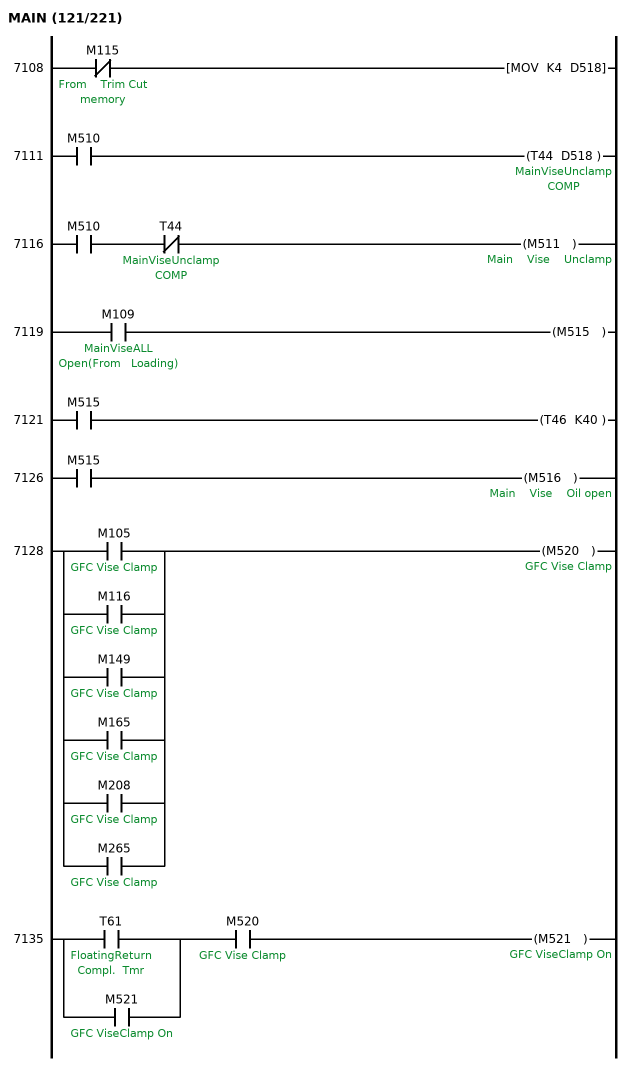
[picture p120: ladder of MAIN, rungs at steps 7108 to 7135]
7108  LDI     M115  ; From    Trim Cut memory
      MOV     K4 D518
7111  LD      M510
      OUT     T44 D518  ; MainViseUnclamp COMP
7116  LD      M510
      ANI     T44  ; MainViseUnclamp COMP
      OUT     M511  ; Main    Vise    Unclamp
7119  LD      M109  ; MainViseALL Open(From   Loading)
      OUT     M515
7121  LD      M515
      OUT     T46 K40
7126  LD      M515
      OUT     M516  ; Main    Vise    Oil open
7128  LD      M105  ; GFC Vise Clamp
      OR      M116  ; GFC Vise Clamp
      OR      M149  ; GFC Vise Clamp
      OR      M165  ; GFC Vise Clamp
      OR      M208  ; GFC Vise Clamp
      OR      M265  ; GFC Vise Clamp
      OUT     M520  ; GFC Vise Clamp
7135  LD      T61  ; FloatingReturn  Compl.  Tmr
      OR      M521  ; GFC ViseClamp On
      AND     M520  ; GFC Vise Clamp
      OUT     M521  ; GFC ViseClamp On
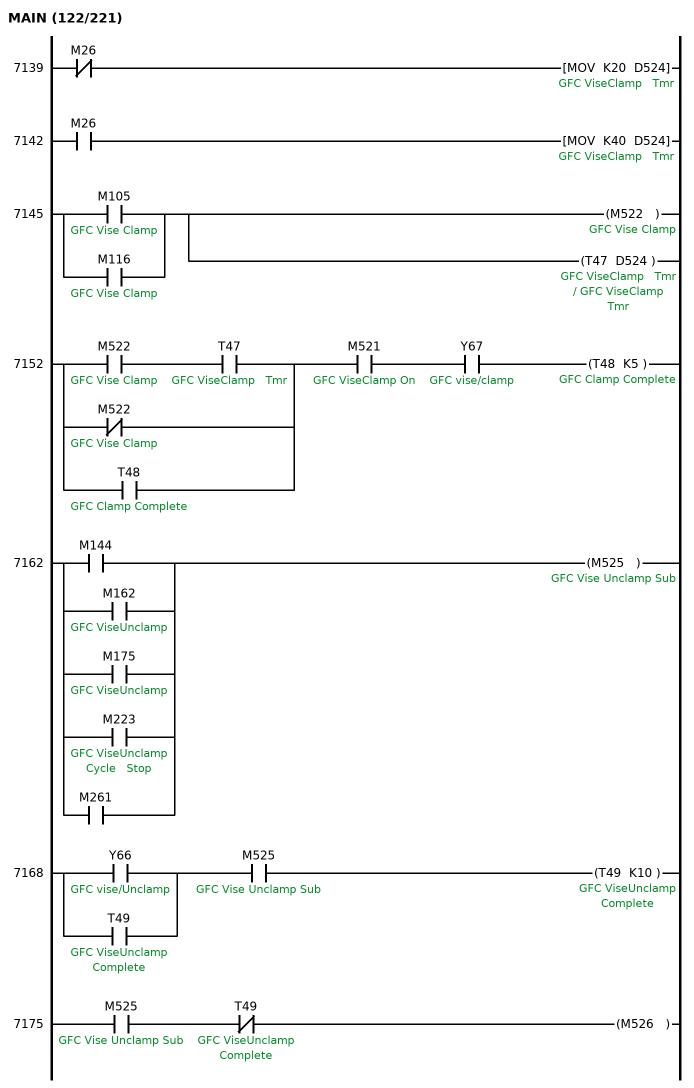
7139  LDI     M26
      MOV     K20 D524  ; GFC ViseClamp   Tmr
7142  LD      M26
      MOV     K40 D524
7145  LD      M105  ; GFC Vise Clamp
      OR      M116  ; GFC Vise Clamp
      OUT     M522  ; GFC Vise Clamp
      OUT     T47 D524  ; GFC ViseClamp   Tmr / GFC ViseClamp   Tmr
7152  LD      M522  ; GFC Vise Clamp
      AND     T47  ; GFC ViseClamp   Tmr
      ORI     M522  ; GFC Vise Clamp
      OR      T48  ; GFC Clamp Complete
      AND     M521  ; GFC ViseClamp On
      AND     Y67  ; GFC vise/clamp
      OUT     T48 K5  ; GFC Clamp Complete
7162  LD      M144
      OR      M162  ; GFC ViseUnclamp
      OR      M175  ; GFC ViseUnclamp
      OR      M223  ; GFC ViseUnclamp Cycle   Stop
      OR      M261
      OUT     M525  ; GFC Vise Unclamp Sub
7168  LD      Y66  ; GFC vise/Unclamp
      OR      T49  ; GFC ViseUnclamp Complete
      AND     M525  ; GFC Vise Unclamp Sub
      OUT     T49 K10  ; GFC ViseUnclamp Complete
7175  LD      M525  ; GFC Vise Unclamp Sub
      ANI     T49  ; GFC ViseUnclamp Complete
      OUT     M526
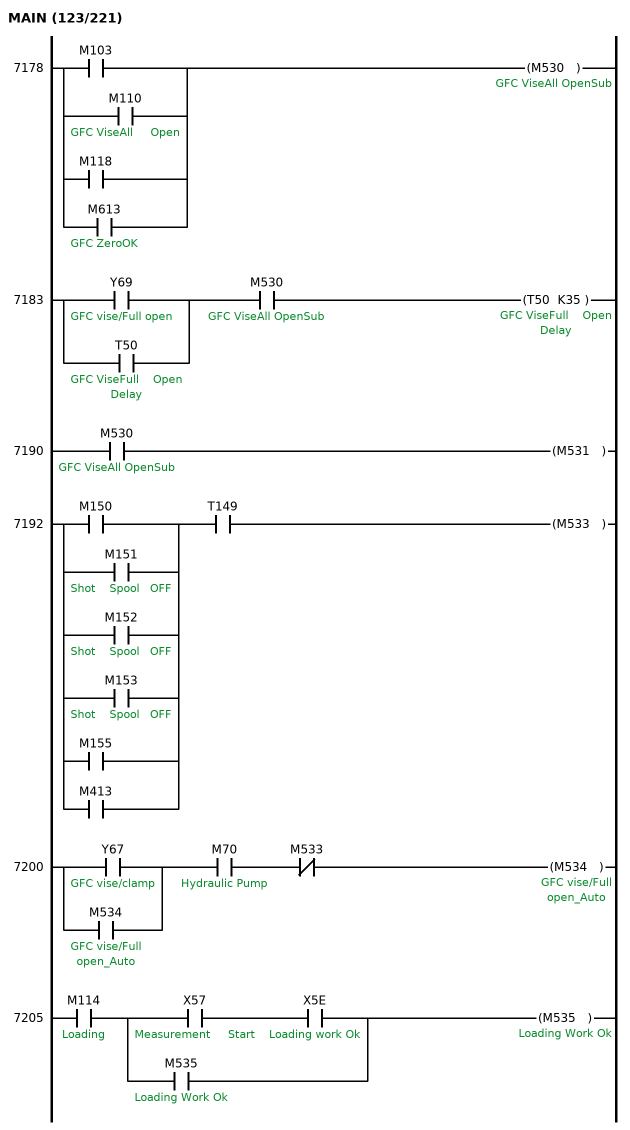
7178  LD      M103
      OR      M110  ; GFC ViseAll     Open
      OR      M118
      OR      M613  ; GFC ZeroOK
      OUT     M530  ; GFC ViseAll OpenSub
7183  LD      Y69  ; GFC vise/Full open
      OR      T50  ; GFC ViseFull    Open    Delay
      AND     M530  ; GFC ViseAll OpenSub
      OUT     T50 K35  ; GFC ViseFull    Open    Delay
7190  LD      M530  ; GFC ViseAll OpenSub
      OUT     M531
7192  LD      M150
      OR      M151  ; Shot    Spool   OFF
      OR      M152  ; Shot    Spool   OFF
      OR      M153  ; Shot    Spool   OFF
      OR      M155
      OR      M413
      AND     T149
      OUT     M533
7200  LD      Y67  ; GFC vise/clamp
      OR      M534  ; GFC vise/Full open_Auto
      AND     M70  ; Hydraulic Pump
      ANI     M533
      OUT     M534  ; GFC vise/Full open_Auto
7205  LD      M114  ; Loading
      LD      X57  ; Measurement     Start
      AND     X5E  ; Loading work Ok
      OR      M535  ; Loading Work Ok
      ANB
      OUT     M535  ; Loading Work Ok
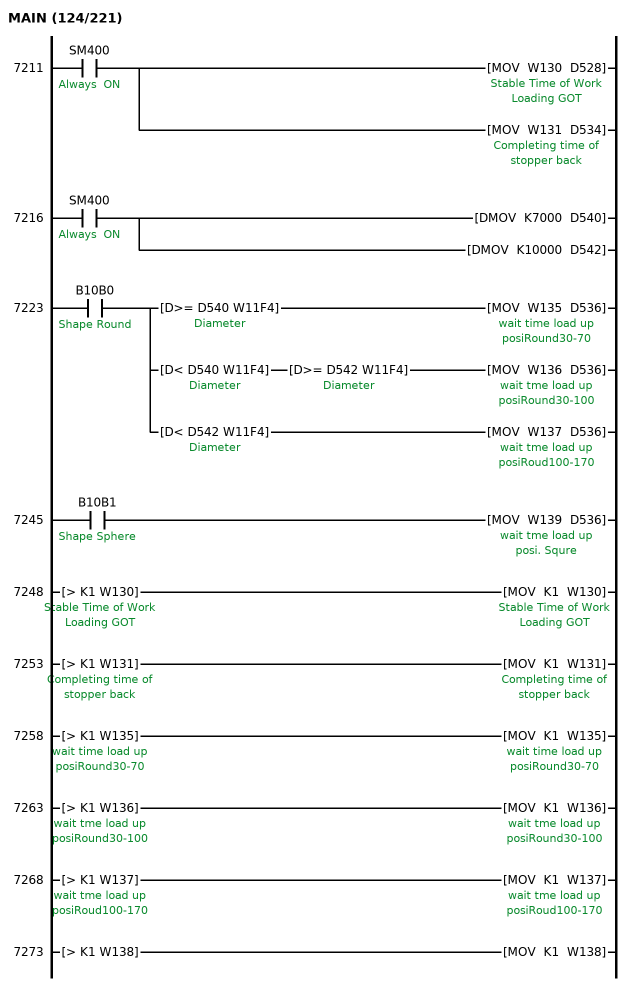
7211  LD      SM400  ; Always  ON
      MOV     W130 D528
      MOV     W131 D534  ; Completing time of stopper back
7216  LD      SM400  ; Always  ON
      DMOV    K7000 D540
      DMOV    K10000 D542
7223  LD      B10B0  ; Shape Round
      MPS
      ANDD>=  D540 W11F4  ; Diameter
      MOV     W135 D536  ; wait time load up posiRound30-70
      MRD
      ANDD<   D540 W11F4  ; Diameter
      ANDD>=  D542 W11F4  ; Diameter
      MOV     W136 D536  ; wait tme load up posiRound30-100
      MPP
      ANDD<   D542 W11F4  ; Diameter
      MOV     W137 D536  ; wait tme load up posiRoud100-170
7245  LD      B10B1  ; Shape Sphere
      MOV     W139 D536  ; wait tme load up posi. Squre
7248  LD>     K1 W130  ; Stable Time of Work Loading GOT
      MOV     K1 W130
7253  LD>     K1 W131  ; Completing time of stopper back
      MOV     K1 W131
7258  LD>     K1 W135  ; wait time load up posiRound30-70
      MOV     K1 W135
7263  LD>     K1 W136  ; wait tme load up posiRound30-100
      MOV     K1 W136
7268  LD>     K1 W137  ; wait tme load up posiRoud100-170
      MOV     K1 W137
7273  LD>     K1 W138
      MOV     K1 W138
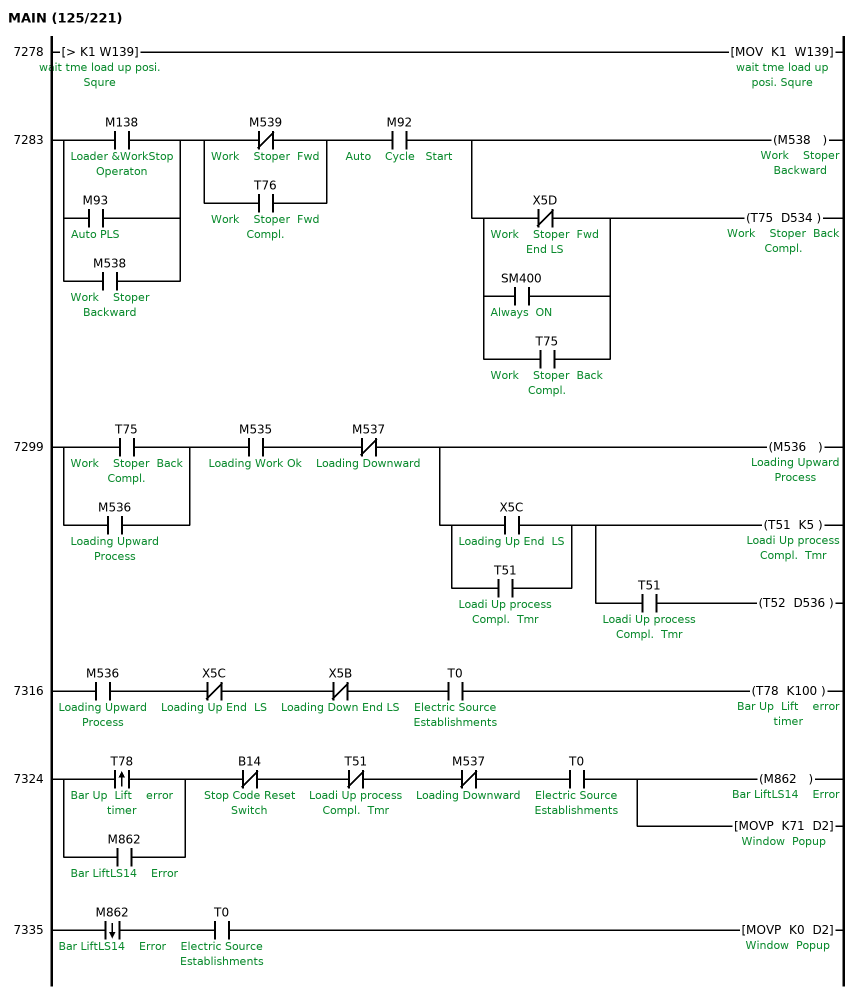
7278  LD>     K1 W139  ; wait tme load up posi. Squre
      MOV     K1 W139
7283  LD      M138  ; Loader &WorkStopOperaton
      OR      M93  ; Auto PLS
      OR      M538  ; Work    Stoper  Backward
      LDI     M539  ; Work    Stoper  Fwd
      OR      T76  ; Work    Stoper  Fwd     Compl.
      ANB
      AND     M92  ; Auto    Cycle   Start
      OUT     M538  ; Work    Stoper  Backward
      LDI     X5D  ; Work    Stoper  Fwd End LS
      OR      SM400  ; Always  ON
      OR      T75  ; Work    Stoper  Back    Compl.
      ANB
      OUT     T75 D534  ; Work    Stoper  Back    Compl.
7299  LD      T75  ; Work    Stoper  Back    Compl.
      OR      M536  ; Loading Upward  Process
      AND     M535  ; Loading Work Ok
      ANI     M537  ; Loading Downward
      OUT     M536  ; Loading Upward  Process
      LD      X5C  ; Loading Up End  LS
      OR      T51  ; Loadi Up process Compl.  Tmr
      ANB
      OUT     T51 K5  ; Loadi Up process Compl.  Tmr
      AND     T51  ; Loadi Up process Compl.  Tmr
      OUT     T52 D536
7316  LD      M536  ; Loading Upward  Process
      ANI     X5C  ; Loading Up End  LS
      ANI     X5B  ; Loading Down End LS
      AND     T0  ; Electric Source Establishments
      OUT     T78 K100  ; Bar Up  Lift    error   timer
7324  LDP     T78  ; Bar Up  Lift    error   timer
      OR      M862  ; Bar LiftLS14    Error
      ANI     B14  ; Stop Code Reset Switch
      ANI     T51  ; Loadi Up process Compl.  Tmr
      ANI     M537  ; Loading Downward
      AND     T0  ; Electric Source Establishments
      OUT     M862  ; Bar LiftLS14    Error
      MOVP    K71 D2  ; Window  Popup
7335  LDF     M862  ; Bar LiftLS14    Error
      AND     T0  ; Electric Source Establishments
      MOVP    K0 D2
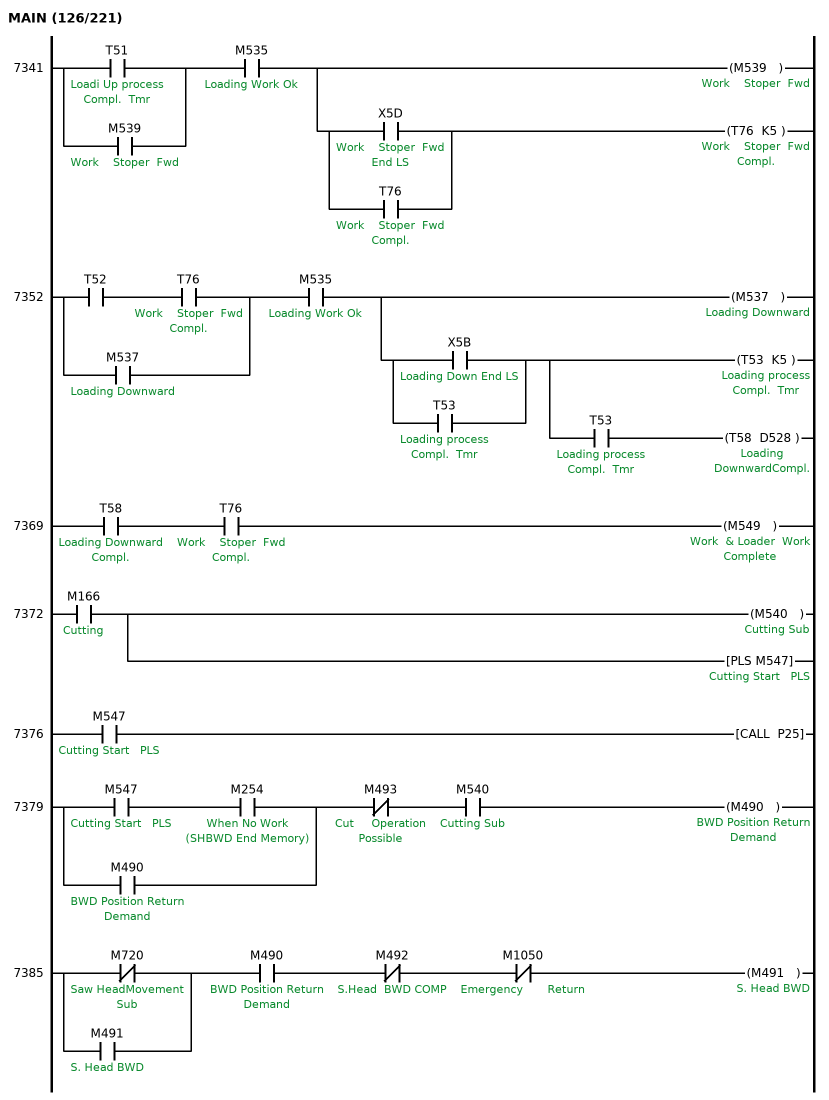
7341  LD      T51  ; Loadi Up process Compl.  Tmr
      OR      M539  ; Work    Stoper  Fwd
      AND     M535  ; Loading Work Ok
      OUT     M539  ; Work    Stoper  Fwd
      LD      X5D  ; Work    Stoper  Fwd End LS
      OR      T76  ; Work    Stoper  Fwd     Compl.
      ANB
      OUT     T76 K5  ; Work    Stoper  Fwd     Compl.
7352  LD      T52
      AND     T76  ; Work    Stoper  Fwd     Compl.
      OR      M537  ; Loading Downward
      AND     M535  ; Loading Work Ok
      OUT     M537  ; Loading Downward
      LD      X5B  ; Loading Down End LS
      OR      T53  ; Loading process Compl.  Tmr
      ANB
      OUT     T53 K5  ; Loading process Compl.  Tmr
      AND     T53  ; Loading process Compl.  Tmr
      OUT     T58 D528  ; Loading DownwardCompl.
7369  LD      T58  ; Loading DownwardCompl.
      AND     T76  ; Work    Stoper  Fwd     Compl.
      OUT     M549  ; Work  & Loader  Work Complete
7372  LD      M166  ; Cutting
      OUT     M540  ; Cutting Sub
      PLS     M547  ; Cutting Start   PLS
7376  LD      M547  ; Cutting Start   PLS
      CALL    P25
7379  LD      M547  ; Cutting Start   PLS
      AND     M254  ; When No Work (SHBWD End Memory)
      OR      M490  ; BWD Position Return Demand
      ANI     M493  ; Cut     Operation       Possible
      AND     M540  ; Cutting Sub
      OUT     M490  ; BWD Position Return Demand
7385  LDI     M720  ; Saw HeadMovementSub
      OR      M491  ; S. Head BWD
      AND     M490  ; BWD Position Return Demand
      ANI     M492  ; S.Head  BWD COMP
      ANI     M1050  ; Emergency       Return
      OUT     M491  ; S. Head BWD
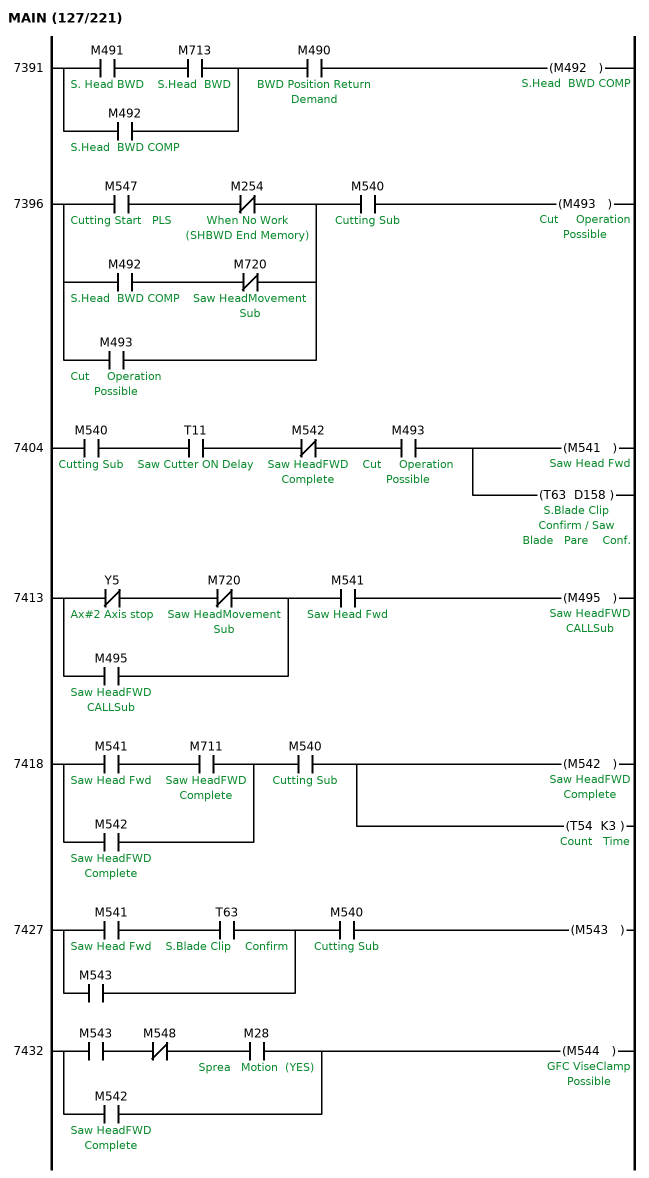
7391  LD      M491  ; S. Head BWD
      AND     M713  ; S.Head  BWD
      OR      M492  ; S.Head  BWD COMP
      AND     M490  ; BWD Position Return Demand
      OUT     M492  ; S.Head  BWD COMP
7396  LD      M547  ; Cutting Start   PLS
      ANI     M254  ; When No Work (SHBWD End Memory)
      LD      M492  ; S.Head  BWD COMP
      ANI     M720  ; Saw HeadMovementSub
      ORB
      OR      M493  ; Cut     Operation       Possible
      AND     M540  ; Cutting Sub
      OUT     M493  ; Cut     Operation       Possible
7404  LD      M540  ; Cutting Sub
      AND     T11  ; Saw Cutter ON Delay
      ANI     M542  ; Saw HeadFWD     Complete
      AND     M493  ; Cut     Operation       Possible
      OUT     M541  ; Saw Head Fwd
      OUT     T63 D158  ; S.Blade Clip    Confirm / Saw     Blade   Pare    Conf.
7413  LDI     Y5  ; Ax#2 Axis stop
      ANI     M720  ; Saw HeadMovementSub
      OR      M495  ; Saw HeadFWD CALLSub
      AND     M541  ; Saw Head Fwd
      OUT     M495  ; Saw HeadFWD CALLSub
7418  LD      M541  ; Saw Head Fwd
      AND     M711  ; Saw HeadFWD     Complete
      OR      M542  ; Saw HeadFWD     Complete
      AND     M540  ; Cutting Sub
      OUT     M542  ; Saw HeadFWD     Complete
      OUT     T54 K3  ; Count   Time
7427  LD      M541  ; Saw Head Fwd
      AND     T63  ; S.Blade Clip    Confirm
      OR      M543
      AND     M540  ; Cutting Sub
      OUT     M543
7432  LD      M543
      ANI     M548
      AND     M28  ; Sprea   Motion  (YES)
      OR      M542  ; Saw HeadFWD     Complete
      OUT     M544  ; GFC ViseClamp   Possible
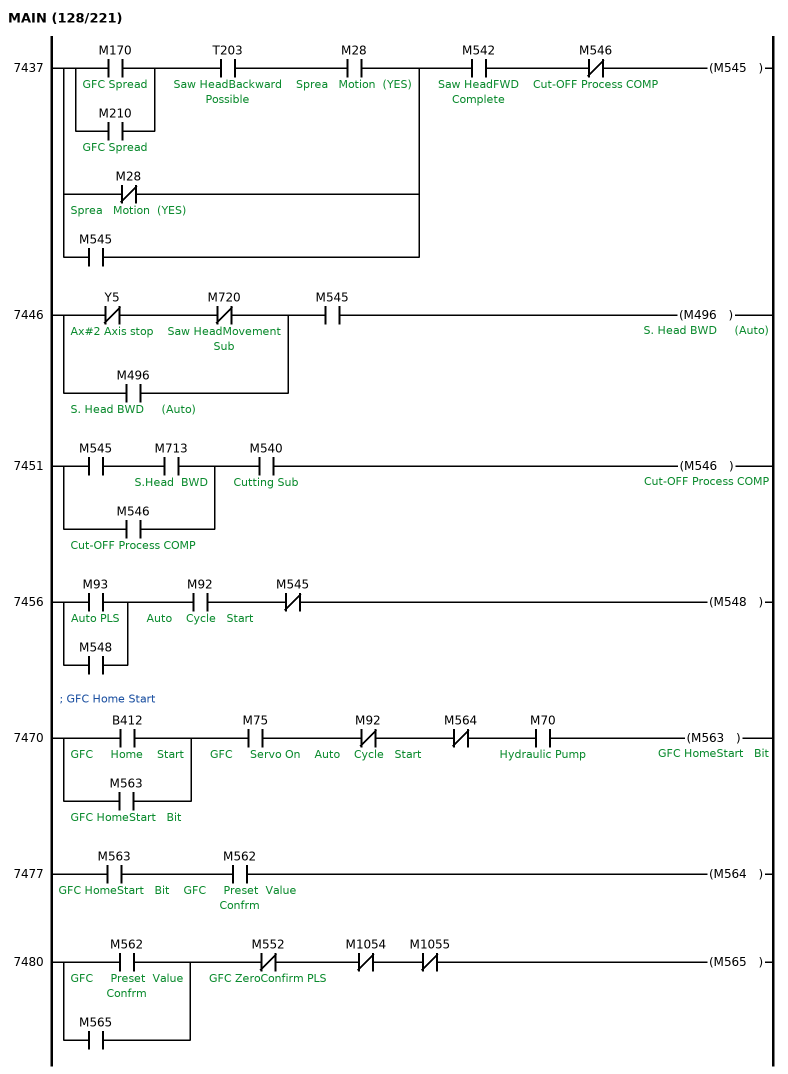
7437  LD      M170  ; GFC Spread
      OR      M210  ; GFC Spread
      AND     T203  ; Saw HeadBackwardPossible
      AND     M28  ; Sprea   Motion  (YES)
      ORI     M28  ; Sprea   Motion  (YES)
      OR      M545
      AND     M542  ; Saw HeadFWD     Complete
      ANI     M546  ; Cut-OFF Process COMP
      OUT     M545
7446  LDI     Y5  ; Ax#2 Axis stop
      ANI     M720  ; Saw HeadMovementSub
      OR      M496  ; S. Head BWD     (Auto)
      AND     M545
      OUT     M496  ; S. Head BWD     (Auto)
7451  LD      M545
      AND     M713  ; S.Head  BWD
      OR      M546  ; Cut-OFF Process COMP
      AND     M540  ; Cutting Sub
      OUT     M546  ; Cut-OFF Process COMP
7456  LD      M93  ; Auto PLS
      OR      M548
      AND     M92  ; Auto    Cycle   Start
      ANI     M545
      OUT     M548
; GFC Home Start
7470  LD      B412  ; GFC     Home    Start
      OR      M563  ; GFC HomeStart   Bit
      AND     M75  ; GFC     Servo On
      ANI     M92  ; Auto    Cycle   Start
      ANI     M564
      AND     M70  ; Hydraulic Pump
      OUT     M563  ; GFC HomeStart   Bit
7477  LD      M563  ; GFC HomeStart   Bit
      AND     M562  ; GFC     Preset  Value   Confrm
      OUT     M564
7480  LD      M562  ; GFC     Preset  Value   Confrm
      OR      M565
      ANI     M552  ; GFC ZeroConfirm PLS
      ANI     M1054
      ANI     M1055
      OUT     M565
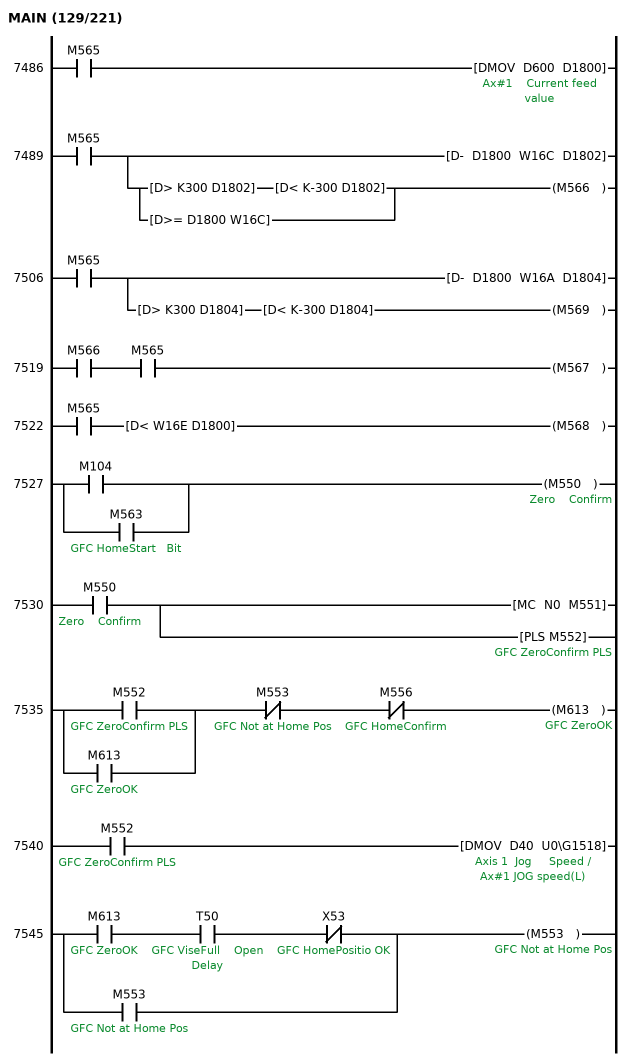
7486  LD      M565
      DMOV    D600 D1800
7489  LD      M565
      D-      D1800 W16C D1802
      LDD>    K300 D1802
      ANDD<   K-300 D1802
      ORD>=   D1800 W16C
      ANB
      OUT     M566
7506  LD      M565
      D-      D1800 W16A D1804
      ANDD>   K300 D1804
      ANDD<   K-300 D1804
      OUT     M569
7519  LD      M566
      AND     M565
      OUT     M567
7522  LD      M565
      ANDD<   W16E D1800
      OUT     M568
7527  LD      M104
      OR      M563  ; GFC HomeStart   Bit
      OUT     M550  ; Zero    Confirm
7530  LD      M550  ; Zero    Confirm
      MC      N0 M551
      PLS     M552  ; GFC ZeroConfirm PLS
7535  LD      M552  ; GFC ZeroConfirm PLS
      OR      M613  ; GFC ZeroOK
      ANI     M553  ; GFC Not at Home Pos
      ANI     M556  ; GFC HomeConfirm
      OUT     M613  ; GFC ZeroOK
7540  LD      M552  ; GFC ZeroConfirm PLS
      DMOV    D40 U0\G1518
7545  LD      M613  ; GFC ZeroOK
      AND     T50  ; GFC ViseFull    Open    Delay
      ANI     X53  ; GFC HomePositio OK
      OR      M553  ; GFC Not at Home Pos
      OUT     M553  ; GFC Not at Home Pos
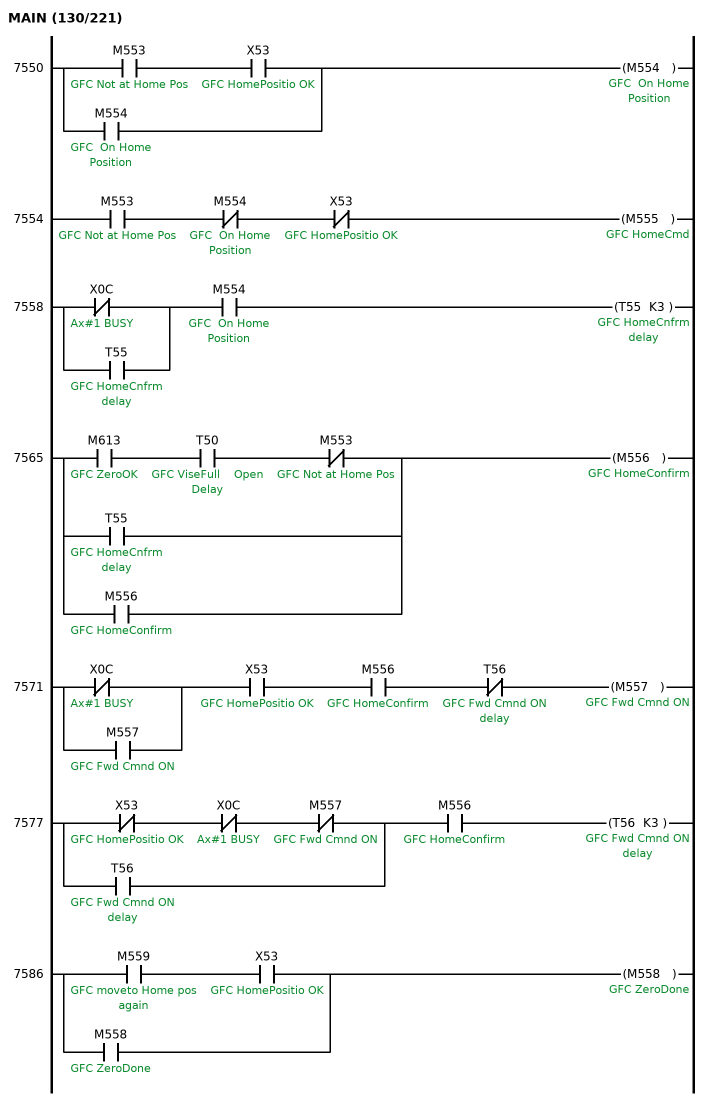
7550  LD      M553  ; GFC Not at Home Pos
      AND     X53  ; GFC HomePositio OK
      OR      M554  ; GFC  On Home    Position
      OUT     M554  ; GFC  On Home    Position
7554  LD      M553  ; GFC Not at Home Pos
      ANI     M554  ; GFC  On Home    Position
      ANI     X53  ; GFC HomePositio OK
      OUT     M555  ; GFC HomeCmd
7558  LDI     X0C  ; Ax#1 BUSY
      OR      T55  ; GFC HomeCnfrm   delay
      AND     M554  ; GFC  On Home    Position
      OUT     T55 K3  ; GFC HomeCnfrm   delay
7565  LD      M613  ; GFC ZeroOK
      AND     T50  ; GFC ViseFull    Open    Delay
      ANI     M553  ; GFC Not at Home Pos
      OR      T55  ; GFC HomeCnfrm   delay
      OR      M556  ; GFC HomeConfirm
      OUT     M556  ; GFC HomeConfirm
7571  LDI     X0C  ; Ax#1 BUSY
      OR      M557  ; GFC Fwd Cmnd ON
      AND     X53  ; GFC HomePositio OK
      AND     M556  ; GFC HomeConfirm
      ANI     T56  ; GFC Fwd Cmnd ON delay
      OUT     M557  ; GFC Fwd Cmnd ON
7577  LDI     X53  ; GFC HomePositio OK
      ANI     X0C  ; Ax#1 BUSY
      ANI     M557  ; GFC Fwd Cmnd ON
      OR      T56  ; GFC Fwd Cmnd ON delay
      AND     M556  ; GFC HomeConfirm
      OUT     T56 K3  ; GFC Fwd Cmnd ON delay
7586  LD      M559  ; GFC moveto Home pos     again
      AND     X53  ; GFC HomePositio OK
      OR      M558  ; GFC ZeroDone
      OUT     M558  ; GFC ZeroDone
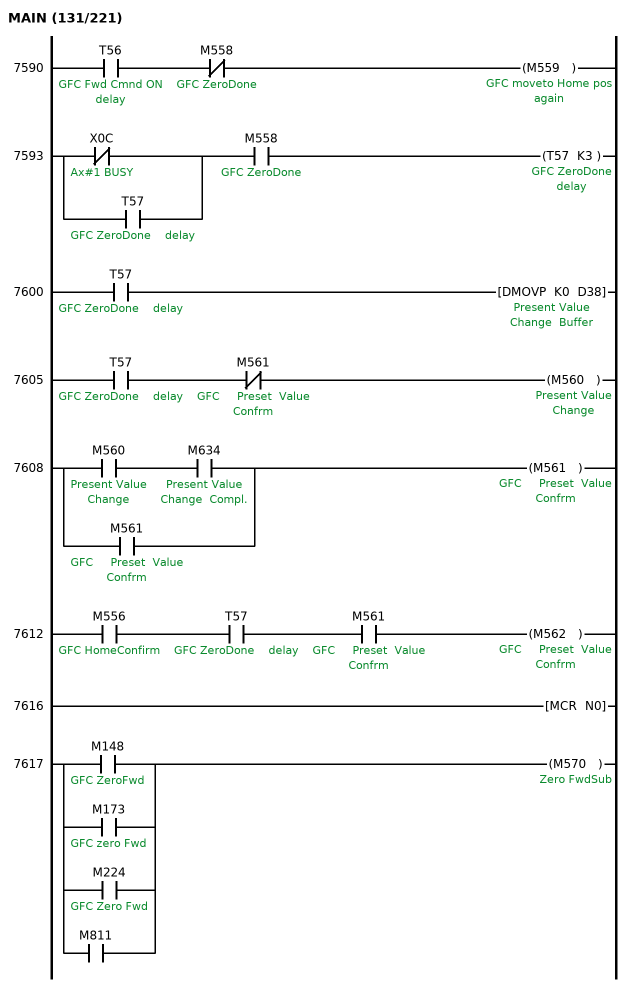
7590  LD      T56  ; GFC Fwd Cmnd ON delay
      ANI     M558  ; GFC ZeroDone
      OUT     M559  ; GFC moveto Home pos     again
7593  LDI     X0C  ; Ax#1 BUSY
      OR      T57  ; GFC ZeroDone    delay
      AND     M558  ; GFC ZeroDone
      OUT     T57 K3  ; GFC ZeroDone    delay
7600  LD      T57  ; GFC ZeroDone    delay
      DMOVP   K0 D38  ; Present Value   Change  Buffer
7605  LD      T57  ; GFC ZeroDone    delay
      ANI     M561  ; GFC     Preset  Value   Confrm
      OUT     M560  ; Present Value   Change
7608  LD      M560  ; Present Value   Change
      AND     M634  ; Present Value   Change  Compl.
      OR      M561  ; GFC     Preset  Value   Confrm
      OUT     M561  ; GFC     Preset  Value   Confrm
7612  LD      M556  ; GFC HomeConfirm
      AND     T57  ; GFC ZeroDone    delay
      AND     M561  ; GFC     Preset  Value   Confrm
      OUT     M562  ; GFC     Preset  Value   Confrm
7616  MCR     N0
7617  LD      M148  ; GFC ZeroFwd
      OR      M173  ; GFC zero Fwd
      OR      M224  ; GFC Zero Fwd
      OR      M811
      OUT     M570  ; Zero FwdSub
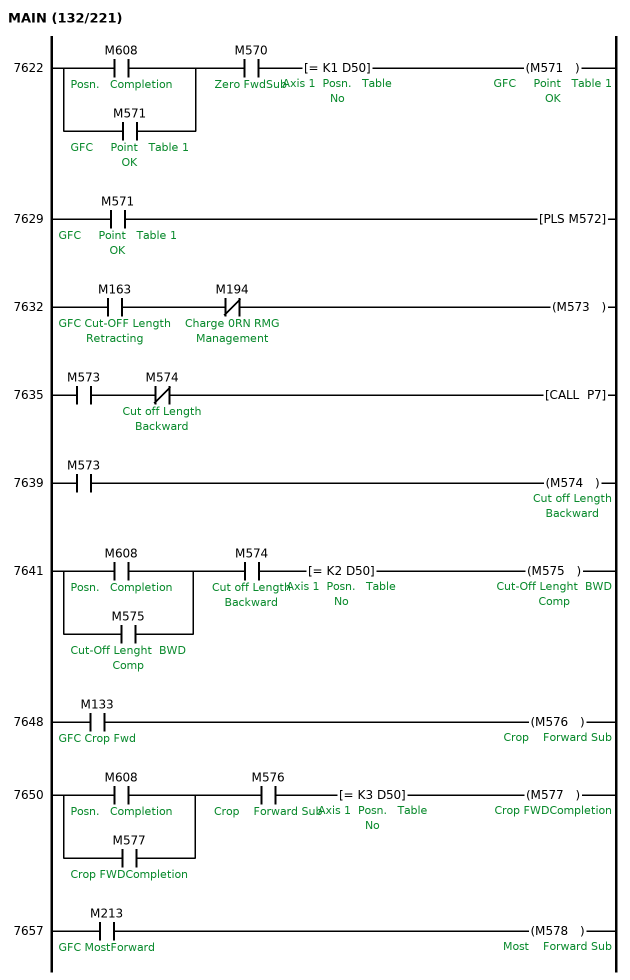
7622  LD      M608  ; Posn.   Completion
      OR      M571  ; GFC     Point   Table 1 OK
      AND     M570  ; Zero FwdSub
      AND=    K1 D50  ; Axis 1  Posn.   Table No
      OUT     M571  ; GFC     Point   Table 1 OK
7629  LD      M571  ; GFC     Point   Table 1 OK
      PLS     M572
7632  LD      M163  ; GFC Cut-OFF Length Retracting
      ANI     M194  ; Charge 0RN RMG  Management
      OUT     M573
7635  LD      M573
      ANI     M574  ; Cut off Length  Backward
      CALL    P7
7639  LD      M573
      OUT     M574  ; Cut off Length  Backward
7641  LD      M608  ; Posn.   Completion
      OR      M575  ; Cut-Off Lenght  BWD Comp
      AND     M574  ; Cut off Length  Backward
      AND=    K2 D50  ; Axis 1  Posn.   Table No
      OUT     M575  ; Cut-Off Lenght  BWD Comp
7648  LD      M133  ; GFC Crop Fwd
      OUT     M576  ; Crop    Forward Sub
7650  LD      M608  ; Posn.   Completion
      OR      M577  ; Crop FWDCompletion
      AND     M576  ; Crop    Forward Sub
      AND=    K3 D50  ; Axis 1  Posn.   Table No
      OUT     M577  ; Crop FWDCompletion
7657  LD      M213  ; GFC MostForward
      OUT     M578  ; Most    Forward Sub
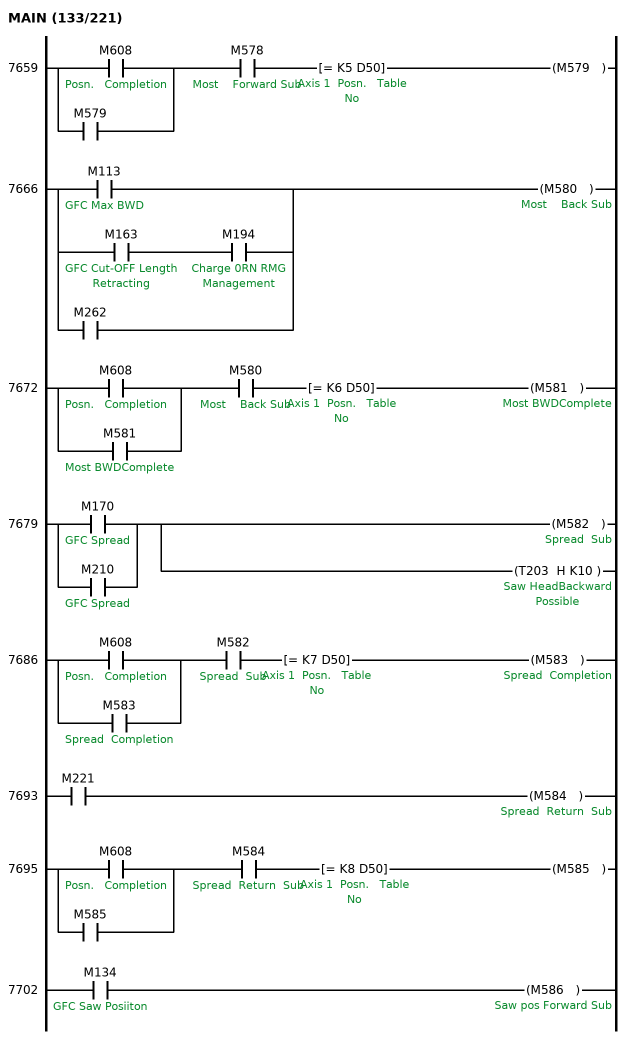
7659  LD      M608  ; Posn.   Completion
      OR      M579
      AND     M578  ; Most    Forward Sub
      AND=    K5 D50  ; Axis 1  Posn.   Table No
      OUT     M579
7666  LD      M113  ; GFC Max BWD
      LD      M163  ; GFC Cut-OFF Length Retracting
      AND     M194  ; Charge 0RN RMG  Management
      ORB
      OR      M262
      OUT     M580  ; Most    Back Sub
7672  LD      M608  ; Posn.   Completion
      OR      M581  ; Most BWDComplete
      AND     M580  ; Most    Back Sub
      AND=    K6 D50  ; Axis 1  Posn.   Table No
      OUT     M581  ; Most BWDComplete
7679  LD      M170  ; GFC Spread
      OR      M210  ; GFC Spread
      OUT     M582  ; Spread  Sub
      OUTH    T203 K10  ; Saw HeadBackwardPossible
7686  LD      M608  ; Posn.   Completion
      OR      M583  ; Spread  Completion
      AND     M582  ; Spread  Sub
      AND=    K7 D50  ; Axis 1  Posn.   Table No
      OUT     M583  ; Spread  Completion
7693  LD      M221
      OUT     M584  ; Spread  Return  Sub
7695  LD      M608  ; Posn.   Completion
      OR      M585
      AND     M584  ; Spread  Return  Sub
      AND=    K8 D50  ; Axis 1  Posn.   Table No
      OUT     M585
7702  LD      M134  ; GFC Saw Posiiton
      OUT     M586  ; Saw pos Forward Sub
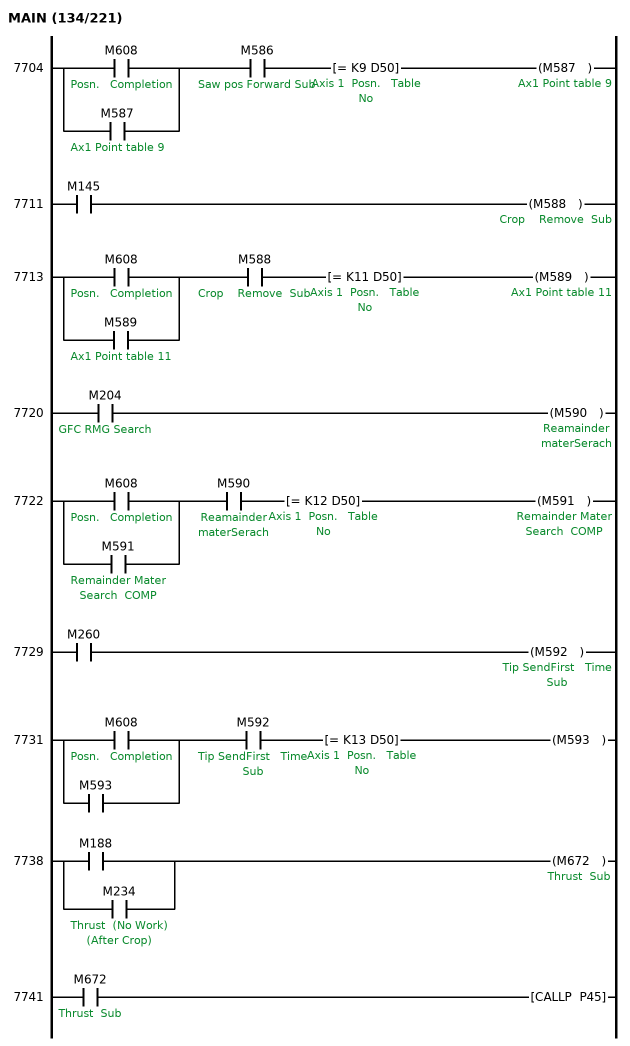
7704  LD      M608  ; Posn.   Completion
      OR      M587  ; Ax1 Point table 9
      AND     M586  ; Saw pos Forward Sub
      AND=    K9 D50  ; Axis 1  Posn.   Table No
      OUT     M587  ; Ax1 Point table 9
7711  LD      M145
      OUT     M588  ; Crop    Remove  Sub
7713  LD      M608  ; Posn.   Completion
      OR      M589  ; Ax1 Point table 11
      AND     M588  ; Crop    Remove  Sub
      AND=    K11 D50  ; Axis 1  Posn.   Table No
      OUT     M589  ; Ax1 Point table 11
7720  LD      M204  ; GFC RMG Search
      OUT     M590  ; Reamainder materSerach
7722  LD      M608  ; Posn.   Completion
      OR      M591  ; Remainder Mater Search  COMP
      AND     M590  ; Reamainder materSerach
      AND=    K12 D50  ; Axis 1  Posn.   Table No
      OUT     M591  ; Remainder Mater Search  COMP
7729  LD      M260
      OUT     M592  ; Tip SendFirst   Time Sub
7731  LD      M608  ; Posn.   Completion
      OR      M593
      AND     M592  ; Tip SendFirst   Time Sub
      AND=    K13 D50  ; Axis 1  Posn.   Table No
      OUT     M593
7738  LD      M188
      OR      M234  ; Thrust  (No Work) (After Crop)
      OUT     M672  ; Thrust  Sub
7741  LD      M672  ; Thrust  Sub
      CALLP   P45
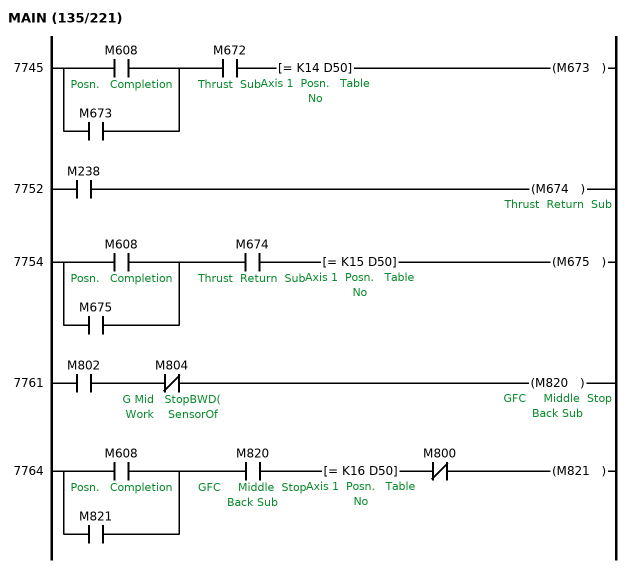
7745  LD      M608  ; Posn.   Completion
      OR      M673
      AND     M672  ; Thrust  Sub
      AND=    K14 D50  ; Axis 1  Posn.   Table No
      OUT     M673
7752  LD      M238
      OUT     M674  ; Thrust  Return  Sub
7754  LD      M608  ; Posn.   Completion
      OR      M675
      AND     M674  ; Thrust  Return  Sub
      AND=    K15 D50  ; Axis 1  Posn.   Table No
      OUT     M675
7761  LD      M802
      ANI     M804  ; G Mid   StopBWD(Work    SensorOf
      OUT     M820  ; GFC     Middle  Stop    Back Sub
7764  LD      M608  ; Posn.   Completion
      OR      M821
      AND     M820  ; GFC     Middle  Stop    Back Sub
      AND=    K16 D50  ; Axis 1  Posn.   Table No
      ANI     M800
      OUT     M821
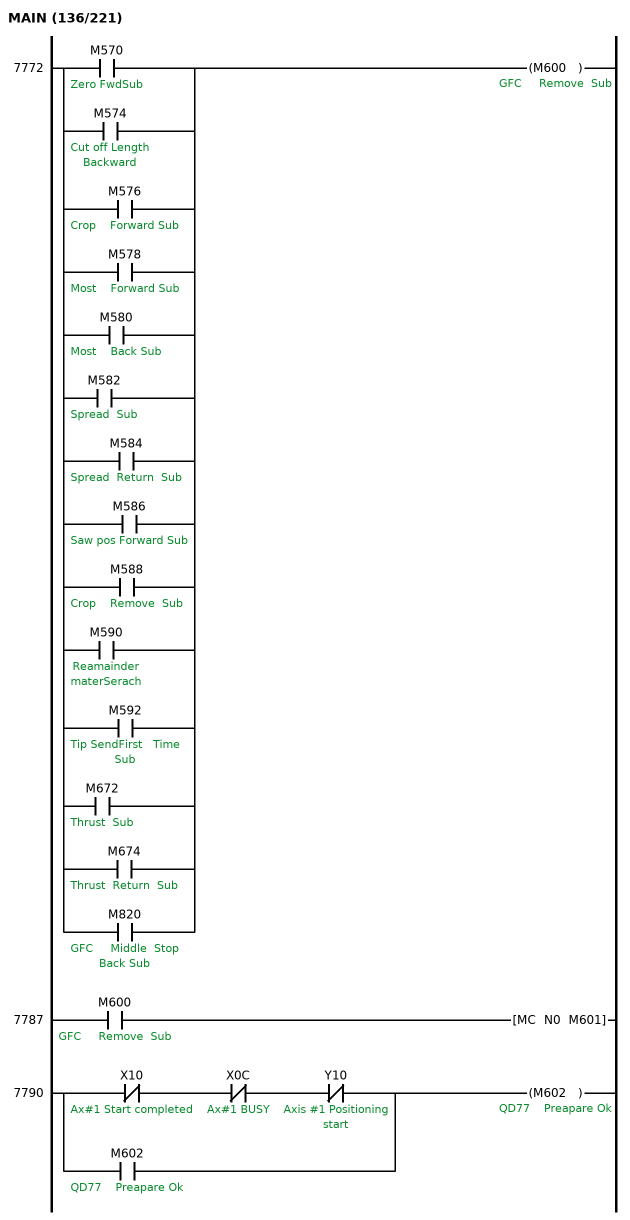
7772  LD      M570  ; Zero FwdSub
      OR      M574  ; Cut off Length  Backward
      OR      M576  ; Crop    Forward Sub
      OR      M578  ; Most    Forward Sub
      OR      M580  ; Most    Back Sub
      OR      M582  ; Spread  Sub
      OR      M584  ; Spread  Return  Sub
      OR      M586  ; Saw pos Forward Sub
      OR      M588  ; Crop    Remove  Sub
      OR      M590  ; Reamainder materSerach
      OR      M592  ; Tip SendFirst   Time Sub
      OR      M672  ; Thrust  Sub
      OR      M674  ; Thrust  Return  Sub
      OR      M820  ; GFC     Middle  Stop    Back Sub
      OUT     M600  ; GFC     Remove  Sub
7787  LD      M600  ; GFC     Remove  Sub
      MC      N0 M601
7790  LDI     X10  ; Ax#1 Start completed
      ANI     X0C  ; Ax#1 BUSY
      ANI     Y10  ; Axis #1 Positioning start
      OR      M602  ; QD77    Preapare Ok
      OUT     M602  ; QD77    Preapare Ok
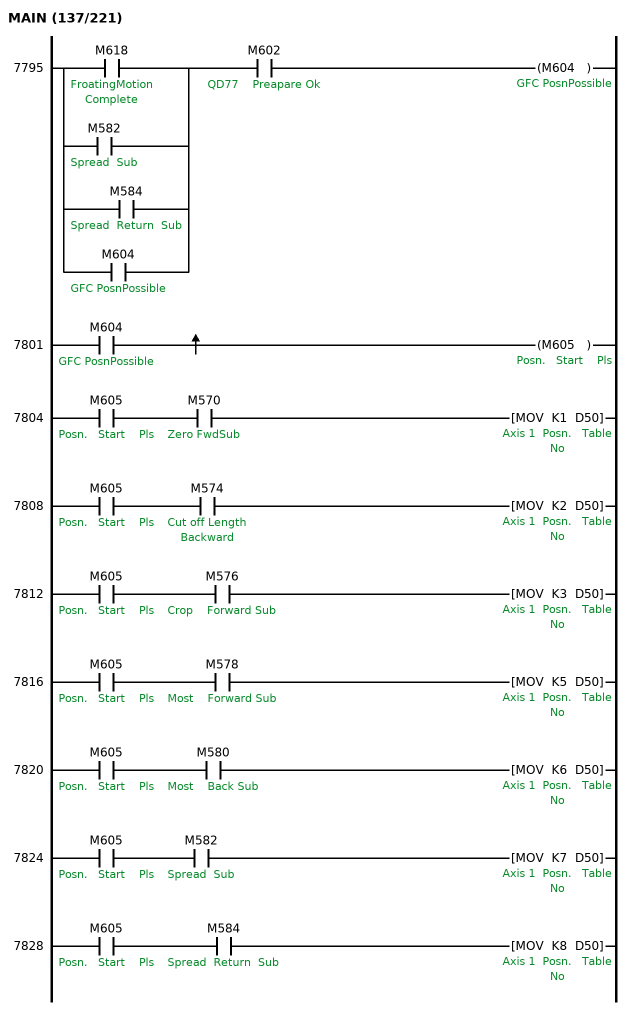
7795  LD      M618  ; FroatingMotion  Complete
      OR      M582  ; Spread  Sub
      OR      M584  ; Spread  Return  Sub
      OR      M604  ; GFC PosnPossible
      AND     M602  ; QD77    Preapare Ok
      OUT     M604  ; GFC PosnPossible
7801  LD      M604  ; GFC PosnPossible
      MEP
      OUT     M605  ; Posn.   Start    Pls
7804  LD      M605  ; Posn.   Start    Pls
      AND     M570  ; Zero FwdSub
      MOV     K1 D50
7808  LD      M605  ; Posn.   Start    Pls
      AND     M574  ; Cut off Length  Backward
      MOV     K2 D50
7812  LD      M605  ; Posn.   Start    Pls
      AND     M576  ; Crop    Forward Sub
      MOV     K3 D50
7816  LD      M605  ; Posn.   Start    Pls
      AND     M578  ; Most    Forward Sub
      MOV     K5 D50
7820  LD      M605  ; Posn.   Start    Pls
      AND     M580  ; Most    Back Sub
      MOV     K6 D50
7824  LD      M605  ; Posn.   Start    Pls
      AND     M582  ; Spread  Sub
      MOV     K7 D50
7828  LD      M605  ; Posn.   Start    Pls
      AND     M584  ; Spread  Return  Sub
      MOV     K8 D50
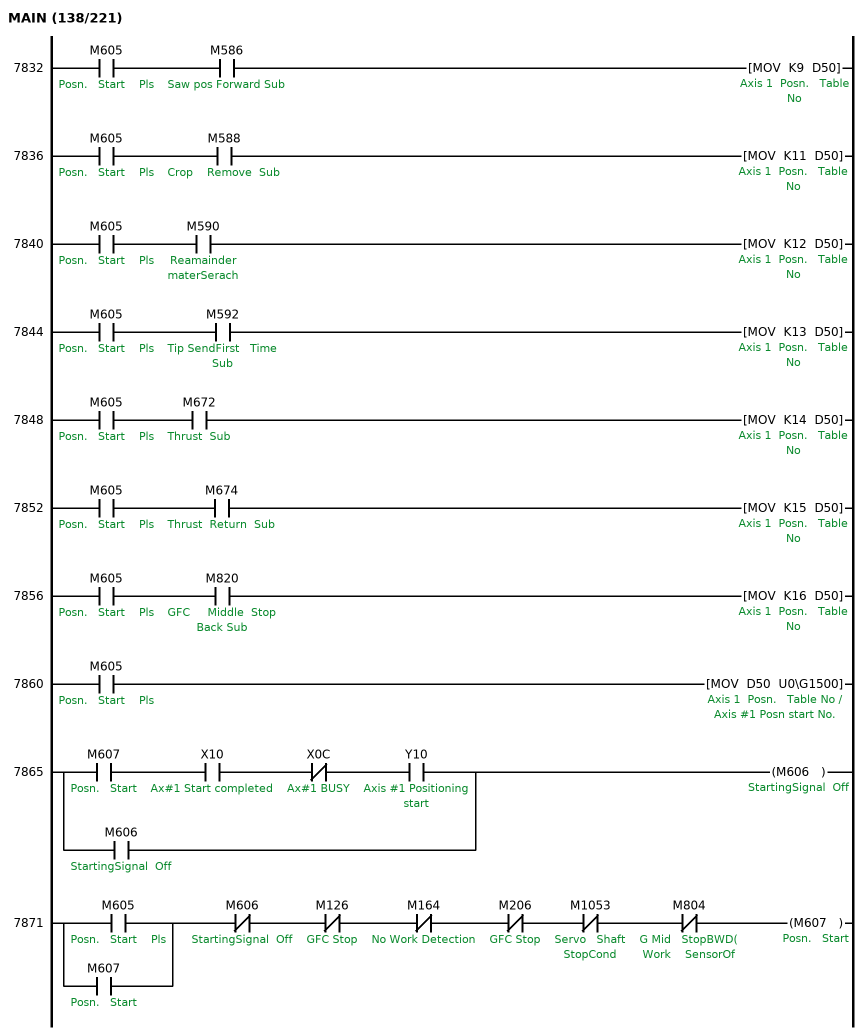
7832  LD      M605  ; Posn.   Start    Pls
      AND     M586  ; Saw pos Forward Sub
      MOV     K9 D50
7836  LD      M605  ; Posn.   Start    Pls
      AND     M588  ; Crop    Remove  Sub
      MOV     K11 D50
7840  LD      M605  ; Posn.   Start    Pls
      AND     M590  ; Reamainder materSerach
      MOV     K12 D50
7844  LD      M605  ; Posn.   Start    Pls
      AND     M592  ; Tip SendFirst   Time Sub
      MOV     K13 D50
7848  LD      M605  ; Posn.   Start    Pls
      AND     M672  ; Thrust  Sub
      MOV     K14 D50
7852  LD      M605  ; Posn.   Start    Pls
      AND     M674  ; Thrust  Return  Sub
      MOV     K15 D50
7856  LD      M605  ; Posn.   Start    Pls
      AND     M820  ; GFC     Middle  Stop    Back Sub
      MOV     K16 D50
7860  LD      M605  ; Posn.   Start    Pls
      MOV     D50 U0\G1500  ; Axis #1 Posn start No.
7865  LD      M607  ; Posn.   Start
      AND     X10  ; Ax#1 Start completed
      ANI     X0C  ; Ax#1 BUSY
      AND     Y10  ; Axis #1 Positioning start
      OR      M606  ; StartingSignal  Off
      OUT     M606  ; StartingSignal  Off
7871  LD      M605  ; Posn.   Start    Pls
      OR      M607  ; Posn.   Start
      ANI     M606  ; StartingSignal  Off
      ANI     M126  ; GFC Stop
      ANI     M164  ; No Work Detection
      ANI     M206  ; GFC Stop
      ANI     M1053  ; Servo   Shaft   StopCond
      ANI     M804  ; G Mid   StopBWD(Work    SensorOf
      OUT     M607  ; Posn.   Start
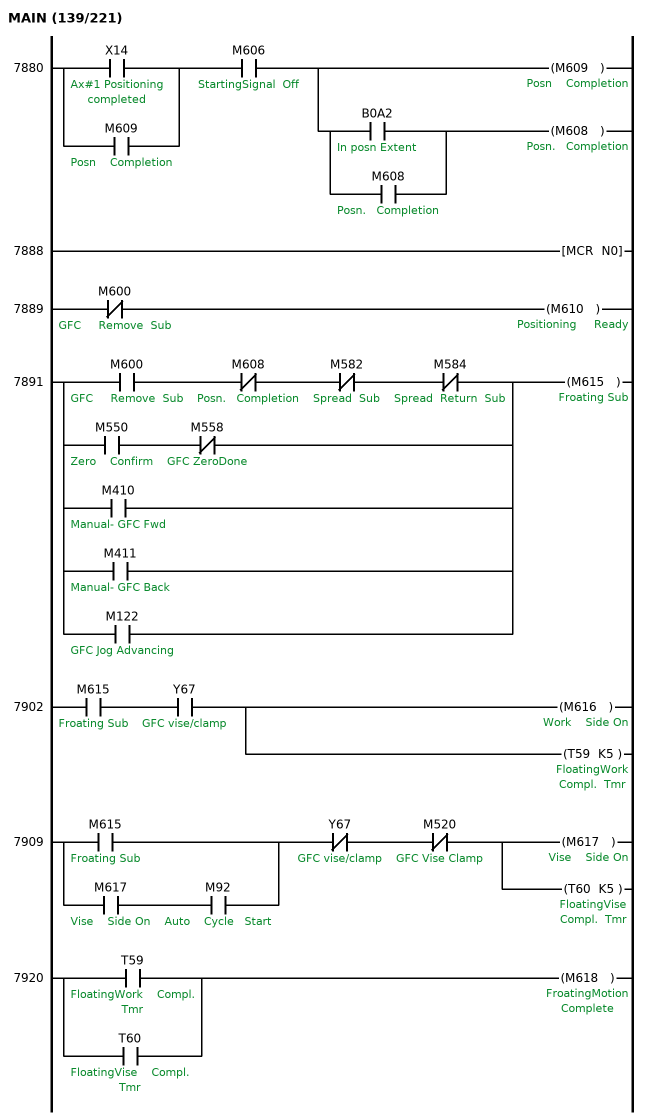
7880  LD      X14  ; Ax#1 Positioning completed
      OR      M609  ; Posn    Completion
      AND     M606  ; StartingSignal  Off
      OUT     M609  ; Posn    Completion
      LD      B0A2  ; In posn Extent
      OR      M608  ; Posn.   Completion
      ANB
      OUT     M608  ; Posn.   Completion
7888  MCR     N0
7889  LDI     M600  ; GFC     Remove  Sub
      OUT     M610  ; Positioning     Ready
7891  LD      M600  ; GFC     Remove  Sub
      ANI     M608  ; Posn.   Completion
      ANI     M582  ; Spread  Sub
      ANI     M584  ; Spread  Return  Sub
      LD      M550  ; Zero    Confirm
      ANI     M558  ; GFC ZeroDone
      ORB
      OR      M410  ; Manual- GFC Fwd
      OR      M411  ; Manual- GFC Back
      OR      M122  ; GFC Jog Advancing
      OUT     M615  ; Froating Sub
7902  LD      M615  ; Froating Sub
      AND     Y67  ; GFC vise/clamp
      OUT     M616  ; Work    Side On
      OUT     T59 K5  ; FloatingWork    Compl.  Tmr
7909  LD      M615  ; Froating Sub
      LD      M617  ; Vise    Side On
      AND     M92  ; Auto    Cycle   Start
      ORB
      ANI     Y67  ; GFC vise/clamp
      ANI     M520  ; GFC Vise Clamp
      OUT     M617  ; Vise    Side On
      OUT     T60 K5  ; FloatingVise    Compl.  Tmr
7920  LD      T59  ; FloatingWork    Compl.  Tmr
      OR      T60  ; FloatingVise    Compl.  Tmr
      OUT     M618  ; FroatingMotion  Complete
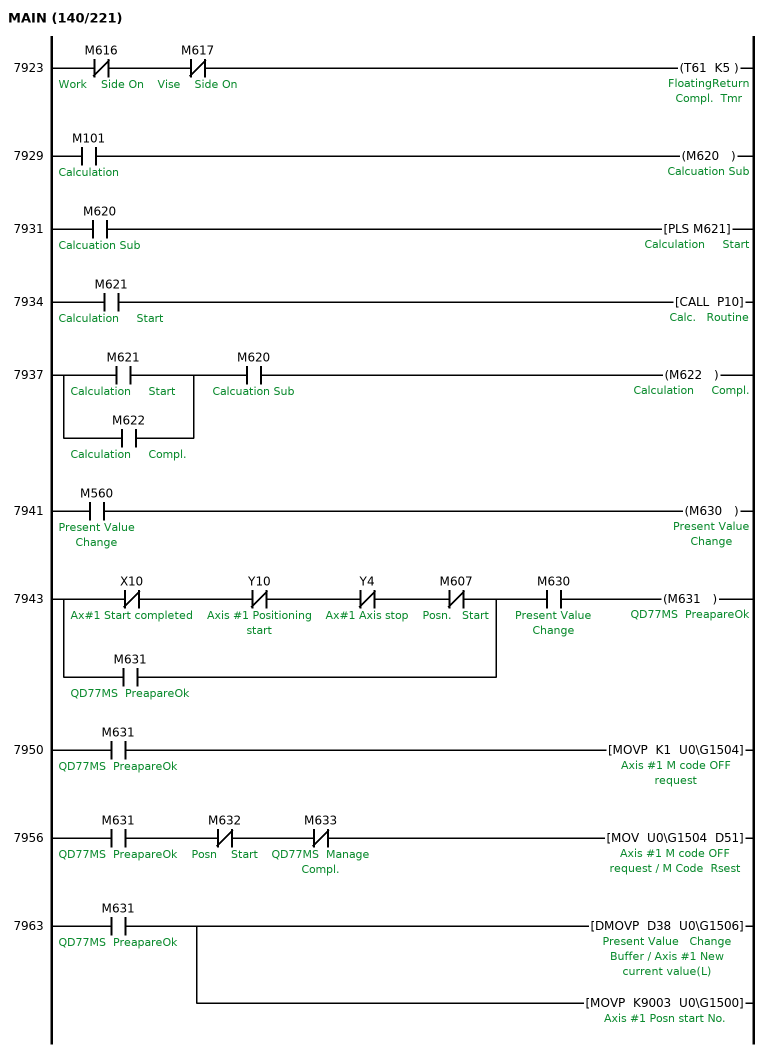
7923  LDI     M616  ; Work    Side On
      ANI     M617  ; Vise    Side On
      OUT     T61 K5  ; FloatingReturn  Compl.  Tmr
7929  LD      M101  ; Calculation
      OUT     M620  ; Calcuation Sub
7931  LD      M620  ; Calcuation Sub
      PLS     M621  ; Calculation     Start
7934  LD      M621  ; Calculation     Start
      CALL    P10  ; Calc.   Routine
7937  LD      M621  ; Calculation     Start
      OR      M622  ; Calculation     Compl.
      AND     M620  ; Calcuation Sub
      OUT     M622  ; Calculation     Compl.
7941  LD      M560  ; Present Value   Change
      OUT     M630  ; Present Value   Change
7943  LDI     X10  ; Ax#1 Start completed
      ANI     Y10  ; Axis #1 Positioning start
      ANI     Y4  ; Ax#1 Axis stop
      ANI     M607  ; Posn.   Start
      OR      M631  ; QD77MS  PreapareOk
      AND     M630  ; Present Value   Change
      OUT     M631  ; QD77MS  PreapareOk
7950  LD      M631  ; QD77MS  PreapareOk
      MOVP    K1 U0\G1504  ; Axis #1 M code OFF request
7956  LD      M631  ; QD77MS  PreapareOk
      ANI     M632  ; Posn    Start
      ANI     M633  ; QD77MS  Manage  Compl.
      MOV     U0\G1504 D51  ; M Code  Rsest
7963  LD      M631  ; QD77MS  PreapareOk
      DMOVP   D38 U0\G1506  ; Axis #1 New current value(L)
      MOVP    K9003 U0\G1500
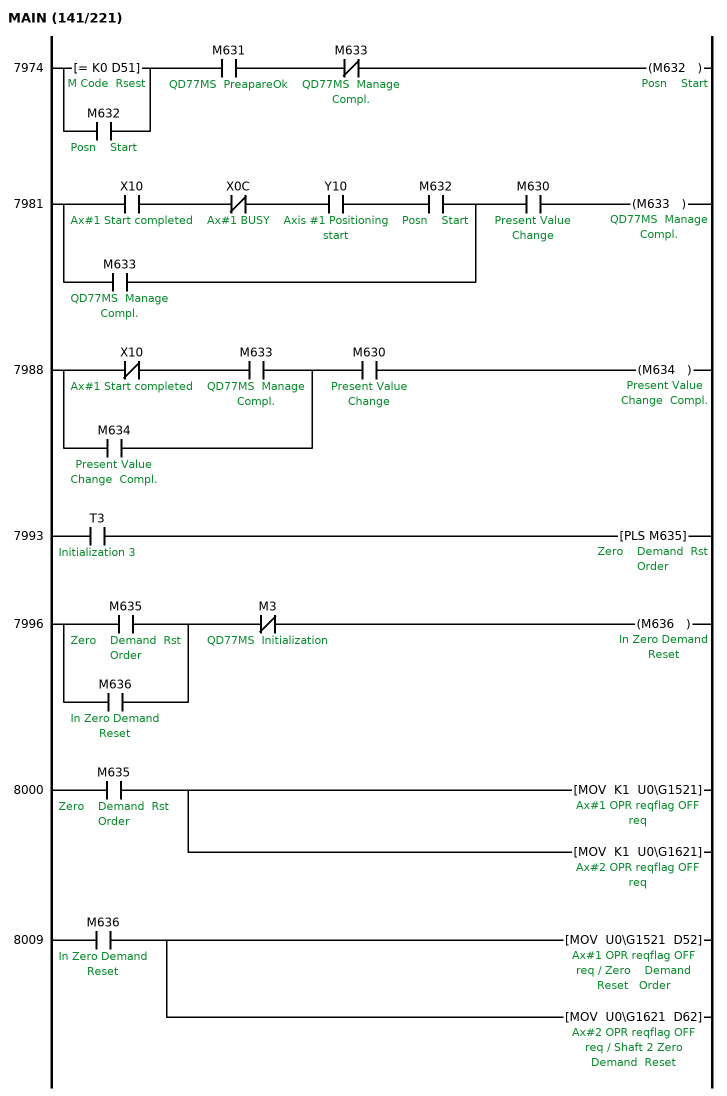
7974  LD=     K0 D51  ; M Code  Rsest
      OR      M632  ; Posn    Start
      AND     M631  ; QD77MS  PreapareOk
      ANI     M633  ; QD77MS  Manage  Compl.
      OUT     M632  ; Posn    Start
7981  LD      X10  ; Ax#1 Start completed
      ANI     X0C  ; Ax#1 BUSY
      AND     Y10  ; Axis #1 Positioning start
      AND     M632  ; Posn    Start
      OR      M633  ; QD77MS  Manage  Compl.
      AND     M630  ; Present Value   Change
      OUT     M633  ; QD77MS  Manage  Compl.
7988  LDI     X10  ; Ax#1 Start completed
      AND     M633  ; QD77MS  Manage  Compl.
      OR      M634  ; Present Value   Change  Compl.
      AND     M630  ; Present Value   Change
      OUT     M634  ; Present Value   Change  Compl.
7993  LD      T3  ; Initialization 3
      PLS     M635  ; Zero    Demand  Rst     Order
7996  LD      M635  ; Zero    Demand  Rst     Order
      OR      M636  ; In Zero Demand  Reset
      ANI     M3  ; QD77MS  Initialization
      OUT     M636  ; In Zero Demand  Reset
8000  LD      M635  ; Zero    Demand  Rst     Order
      MOV     K1 U0\G1521  ; Ax#1 OPR reqflag OFF req
      MOV     K1 U0\G1621  ; Ax#2 OPR reqflag OFF req
8009  LD      M636  ; In Zero Demand  Reset
      MOV     U0\G1521 D52  ; Zero    Demand  Reset   Order
      MOV     U0\G1621 D62  ; Shaft 2 Zero    Demand  Reset
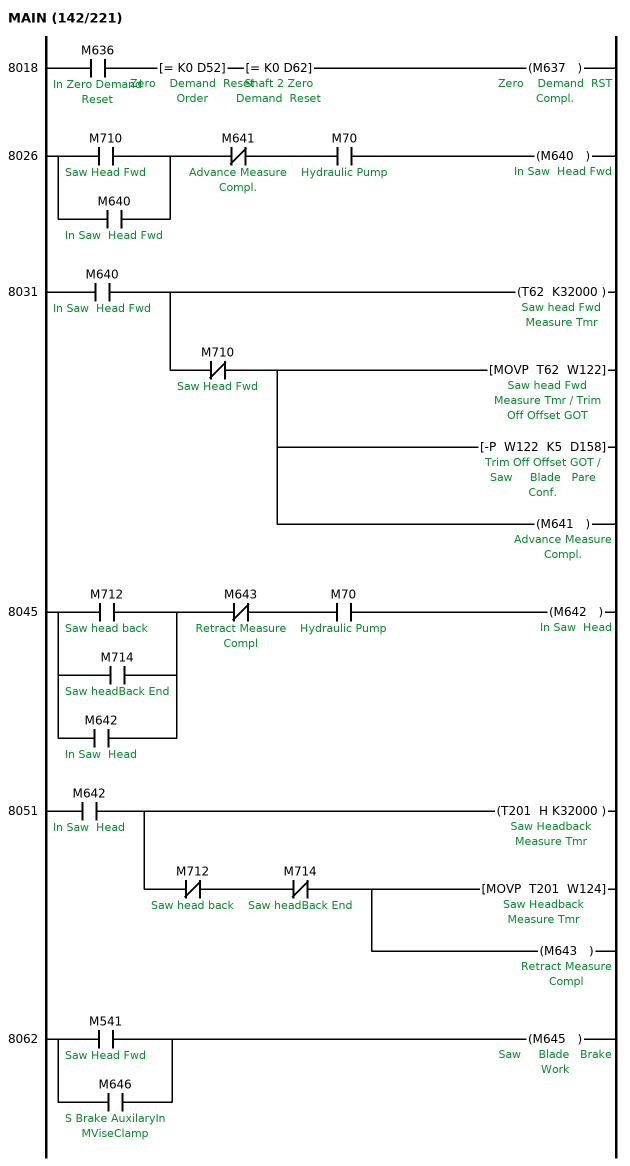
8018  LD      M636  ; In Zero Demand  Reset
      AND=    K0 D52  ; Zero    Demand  Reset   Order
      AND=    K0 D62  ; Shaft 2 Zero    Demand  Reset
      OUT     M637  ; Zero    Demand  RST     Compl.
8026  LD      M710  ; Saw Head Fwd
      OR      M640  ; In Saw  Head Fwd
      ANI     M641  ; Advance Measure Compl.
      AND     M70  ; Hydraulic Pump
      OUT     M640  ; In Saw  Head Fwd
8031  LD      M640  ; In Saw  Head Fwd
      OUT     T62 K32000  ; Saw head Fwd    Measure Tmr
      ANI     M710  ; Saw Head Fwd
      MOVP    T62 W122  ; Trim Off Offset GOT
      -P      W122 K5 D158
      OUT     M641  ; Advance Measure Compl.
8045  LD      M712  ; Saw head back
      OR      M714  ; Saw headBack End
      OR      M642  ; In Saw  Head
      ANI     M643  ; Retract Measure Compl
      AND     M70  ; Hydraulic Pump
      OUT     M642  ; In Saw  Head
8051  LD      M642  ; In Saw  Head
      OUTH    T201 K32000  ; Saw Headback    Measure Tmr
      ANI     M712  ; Saw head back
      ANI     M714  ; Saw headBack End
      MOVP    T201 W124
      OUT     M643  ; Retract Measure Compl
8062  LD      M541  ; Saw Head Fwd
      OR      M646  ; S Brake AuxilaryIn MViseClamp
      OUT     M645  ; Saw     Blade   Brake   Work
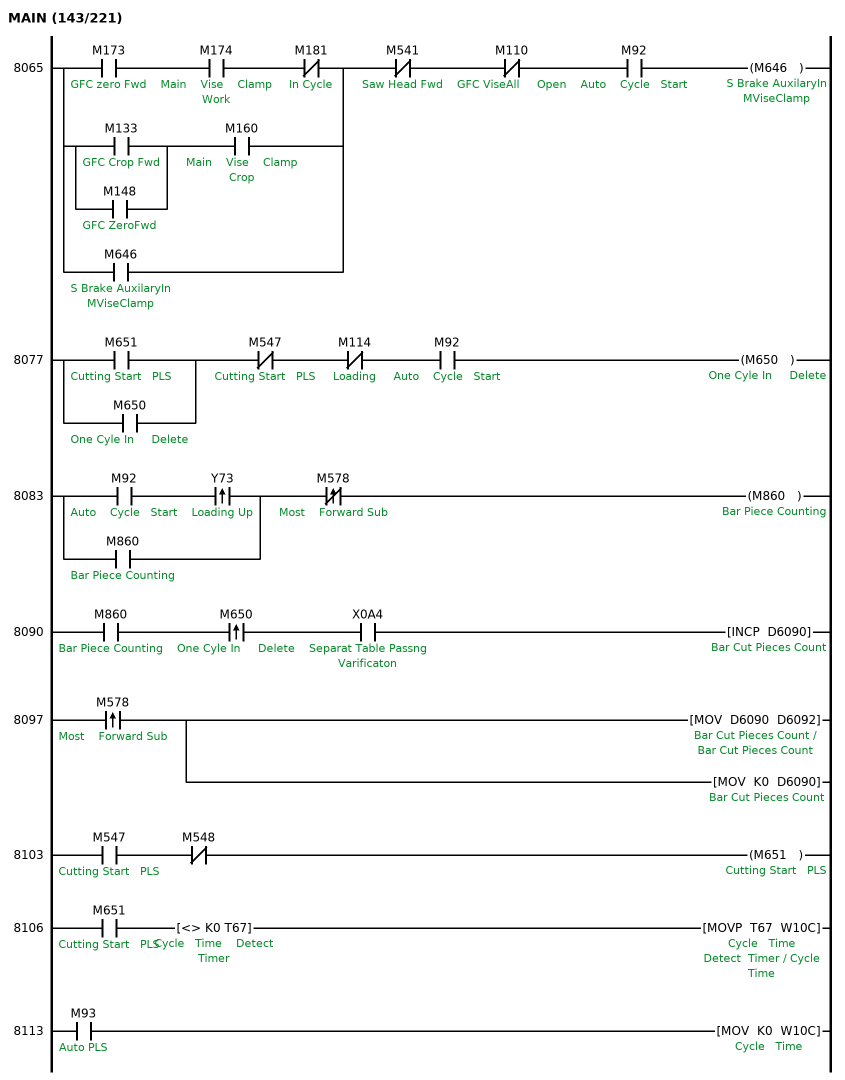
8065  LD      M173  ; GFC zero Fwd
      AND     M174  ; Main    Vise    Clamp   Work
      ANI     M181  ; In Cycle
      LD      M133  ; GFC Crop Fwd
      OR      M148  ; GFC ZeroFwd
      AND     M160  ; Main    Vise    Clamp   Crop
      ORB
      OR      M646  ; S Brake AuxilaryIn MViseClamp
      ANI     M541  ; Saw Head Fwd
      ANI     M110  ; GFC ViseAll     Open
      AND     M92  ; Auto    Cycle   Start
      OUT     M646  ; S Brake AuxilaryIn MViseClamp
8077  LD      M651  ; Cutting Start   PLS
      OR      M650  ; One Cyle In     Delete
      ANI     M547  ; Cutting Start   PLS
      ANI     M114  ; Loading
      AND     M92  ; Auto    Cycle   Start
      OUT     M650  ; One Cyle In     Delete
8083  LD      M92  ; Auto    Cycle   Start
      ANDP    Y73  ; Loading Up
      OR      M860  ; Bar Piece Counting
      ANDPI   M578  ; Most    Forward Sub
      OUT     M860  ; Bar Piece Counting
8090  LD      M860  ; Bar Piece Counting
      ANDP    M650  ; One Cyle In     Delete
      AND     X0A4  ; Separat Table Passng Varificaton
      INCP    D6090  ; Bar Cut Pieces Count
8097  LDP     M578  ; Most    Forward Sub
      MOV     D6090 D6092  ; Bar Cut Pieces Count
      MOV     K0 D6090
8103  LD      M547  ; Cutting Start   PLS
      ANI     M548
      OUT     M651  ; Cutting Start   PLS
8106  LD      M651  ; Cutting Start   PLS
      AND<>   K0 T67  ; Cycle   Time    Detect  Timer
      MOVP    T67 W10C  ; Cycle   Time
8113  LD      M93  ; Auto PLS
      MOV     K0 W10C
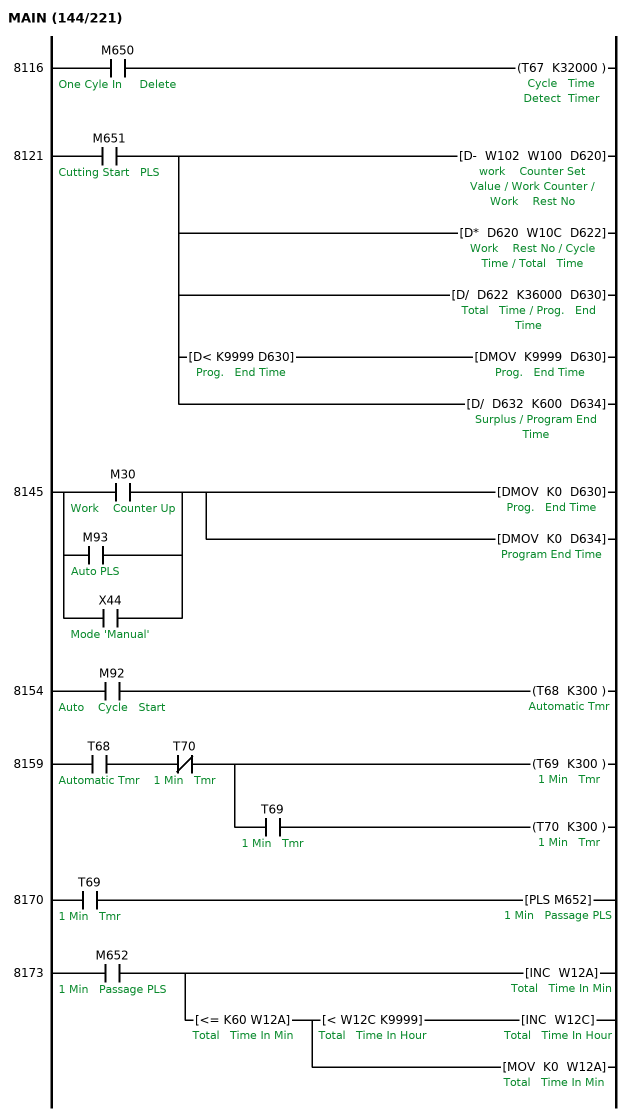
8116  LD      M650  ; One Cyle In     Delete
      OUT     T67 K32000  ; Cycle   Time    Detect  Timer
8121  LD      M651  ; Cutting Start   PLS
      D-      W102 W100 D620  ; Work    Rest No
      D*      D620 W10C D622  ; Total   Time
      D/      D622 K36000 D630  ; Prog.   End Time
      MPS
      ANDD<   K9999 D630  ; Prog.   End Time
      DMOV    K9999 D630
      MPP
      D/      D632 K600 D634  ; Surplus / Program End Time
8145  LD      M30  ; Work    Counter Up
      OR      M93  ; Auto PLS
      OR      X44  ; Mode 'Manual'
      DMOV    K0 D630
      DMOV    K0 D634
8154  LD      M92  ; Auto    Cycle   Start
      OUT     T68 K300  ; Automatic Tmr
8159  LD      T68  ; Automatic Tmr
      ANI     T70  ; 1 Min   Tmr
      OUT     T69 K300  ; 1 Min   Tmr
      AND     T69  ; 1 Min   Tmr
      OUT     T70 K300  ; 1 Min   Tmr
8170  LD      T69  ; 1 Min   Tmr
      PLS     M652  ; 1 Min   Passage PLS
8173  LD      M652  ; 1 Min   Passage PLS
      INC     W12A  ; Total   Time In Min
      AND<=   K60 W12A  ; Total   Time In Min
      MPS
      AND<    W12C K9999  ; Total   Time In Hour
      INC     W12C
      MPP
      MOV     K0 W12A
